{attribute 'qualified_only'}
TYPE E_SerialError :
(
	eNoError := 0,
	eComBufferError,
	eOutputBufferTooSmall,
	eChecksumFailed
);
END_TYPE

(* stored: Version 1.1.0.1, ProductVersion 3.1.4024.9
   DUT E_SerialError: Id {135869b0-a909-4423-8b39-3e668d4613a7} *)
